// TIA Portal V17 export
// export: Created 2024-08-29T18:23:49.4576006Z, ExportSetting WithDefaults, DisplayName Totally Integrated Automation Portal, DisplayVersion V17 Update 7, DisplayName TIA Portal Openness, DisplayVersion V17 Update 7, DisplayName TIA Portal Version Control Interface, DisplayVersion V17, DisplayName SINAMICS Startdrive Advanced, DisplayVersion V17 SP2, DisplayName SINAMICS Startdrive G110M, G120, G120C, G120D, G120P, G115D, DisplayVersion V17 SP2, DisplayName SINAMICS Startdrive G130, G150, S120, S150, SINAMICS MV, S210, DisplayVersion V17 SP2, DisplayName STEP 7 Professional, DisplayVersion V17 Update 7, DisplayName STEP 7 Safety, DisplayVersion V17 Update 6, DisplayName WinCC Advanced / Unified PC, DisplayVersion V17 Update 7
DATA_BLOCK "Receive_Reset_DB2"   // DB39
// stored: AutoNumber true, DBAccessibleFromOPCUA true, DBAccessibleFromWebserver true, InstanceOfName Receive_Reset, OfSystemLibElement Receive_Reset, OfSystemLibVersion 1.2
"Receive_Reset"
   // VAR_INPUT
   //    REQ : Bool := FALSE;
   //    PORT : Word := 16#0132;
   // END_VAR
   // VAR_OUTPUT
   //    DONE : Bool := FALSE;
   //    ERROR : Bool := FALSE;
   //    STATUS : Word := 16#7000;
   // END_VAR
   // VAR
   //    b_e_REQ : Bool := FALSE;
   //    y_state : SInt := 0;
   //    WRREC { S7_SetPoint := 'True'} : WRREC;
   //    w_record { S7_SetPoint := 'True'} : P2P_ResetData;
   // END_VAR
BEGIN
   WRREC.REQ := FALSE;
   WRREC.ID := 306;
   WRREC.INDEX := 54;
   WRREC.LEN := 12;
   WRREC.DONE := TRUE;
   WRREC.BUSY := FALSE;
   WRREC.ERROR := FALSE;
   WRREC.STATUS := 16#0000_0000;
   w_record.header.block_type := 16#0036;
   w_record.header.block_len := 16#0008;
   w_record.header.block_ver := 16#0100;
   w_record.header.res := 16#0000;
   w_record.ackn := 16#01;
   w_record.res1 := 16#00;
   w_record.res2 := 16#00;
   w_record.res3 := 16#00;
END_DATA_BLOCK
